(* CoDeSys 2.3.9.31 project: X758PLC.pro *)
(* Libraries: TcBase.lib 14.5.09 11:14:08, TcSystem.lib 27.2.12 14:08:36, TcBaseMath.lib 27.7.04 11:07:56, TcMath.lib 23.9.04 14:15:30, TcMC2.lib 23.8.12 10:01:14, STANDARD.LIB 5.6.98 11:03:02 *)

(* Task configuration *)
TASK Standard (PRIORITY := 0, INTERVAL := T#10ms);
	MAIN
END_TASK

(* Global variable list: Global_Variables *)
VAR_GLOBAL
	Axis_X	:	Axis_Ref;
	Axis_Y	:	Axis_Ref;
	Axis_F	:	Axis_Ref;
	Axis_T	:	Axis_Ref;
END_VAR

(* Global variable list: TwinCAT_Configuration *)
(* Generated automatically by TwinCAT - (read only) *)
VAR_CONFIG
	MAIN.BFI1 AT %IX512.0 : BOOL;	(*  ~ {LinkedWith:TIID^Device 2 (EtherCAT)^Term 1 (EK1100)^Term 2 (EL1889)^Channel 1^Input} *)
	MAIN.BFI2 AT %IX512.1 : BOOL;	(*  ~ {LinkedWith:TIID^Device 2 (EtherCAT)^Term 1 (EK1100)^Term 2 (EL1889)^Channel 2^Input} *)
	MAIN.BFI3 AT %IX512.2 : BOOL;	(*  ~ {LinkedWith:TIID^Device 2 (EtherCAT)^Term 1 (EK1100)^Term 2 (EL1889)^Channel 3^Input} *)
	MAIN.BFI4 AT %IX512.3 : BOOL;	(*  ~ {LinkedWith:TIID^Device 2 (EtherCAT)^Term 1 (EK1100)^Term 2 (EL1889)^Channel 4^Input} *)
	MAIN.BFI5 AT %IX512.4 : BOOL;	(*  ~ {LinkedWith:TIID^Device 2 (EtherCAT)^Term 1 (EK1100)^Term 2 (EL1889)^Channel 5^Input} *)
	MAIN.BFI6 AT %IX512.5 : BOOL;	(*  ~ {LinkedWith:TIID^Device 2 (EtherCAT)^Term 1 (EK1100)^Term 2 (EL1889)^Channel 6^Input} *)
	MAIN.BFI7 AT %IX512.6 : BOOL;	(*  ~ {LinkedWith:TIID^Device 2 (EtherCAT)^Term 1 (EK1100)^Term 2 (EL1889)^Channel 7^Input} *)
	MAIN.BFI8 AT %IX516.0 : BOOL;
	MAIN.BFI9 AT %IX516.1 : BOOL;
	MAIN.BFO1 AT %QX512.0 : BOOL;	(*  ~ {LinkedWith:TIID^Device 2 (EtherCAT)^Term 1 (EK1100)^Term 3 (EL2889)^Channel 1^Output} *)
	MAIN.BFO2 AT %QX512.1 : BOOL;	(*  ~ {LinkedWith:TIID^Device 2 (EtherCAT)^Term 1 (EK1100)^Term 3 (EL2889)^Channel 2^Output} *)
	MAIN.BFO3 AT %QX512.2 : BOOL;	(*  ~ {LinkedWith:TIID^Device 2 (EtherCAT)^Term 1 (EK1100)^Term 3 (EL2889)^Channel 3^Output} *)
	.Axis_X.PlcToNc AT %QB0 : PLCTONC_AXIS_REF;	(*  ~ {LinkedWith:TINC^NC-Task 1 SAF^Axes^Axis 1^Inputs^Axis 1_FromPlc} *)
	.Axis_X.NcToPlc AT %IB0 : NCTOPLC_AXIS_REF;	(*  ~ {LinkedWith:TINC^NC-Task 1 SAF^Axes^Axis 1^Outputs^Axis 1_ToPlc} *)
	.Axis_Y.PlcToNc AT %QB128 : PLCTONC_AXIS_REF;	(*  ~ {LinkedWith:TINC^NC-Task 1 SAF^Axes^Axis 2^Inputs^Axis 2_FromPlc} *)
	.Axis_Y.NcToPlc AT %IB128 : NCTOPLC_AXIS_REF;	(*  ~ {LinkedWith:TINC^NC-Task 1 SAF^Axes^Axis 2^Outputs^Axis 2_ToPlc} *)
	.Axis_F.PlcToNc AT %QB256 : PLCTONC_AXIS_REF;	(*  ~ {LinkedWith:TINC^NC-Task 1 SAF^Axes^Axis 3^Inputs^Axis 3_FromPlc} *)
	.Axis_F.NcToPlc AT %IB256 : NCTOPLC_AXIS_REF;	(*  ~ {LinkedWith:TINC^NC-Task 1 SAF^Axes^Axis 3^Outputs^Axis 3_ToPlc} *)
	.Axis_T.PlcToNc AT %QB384 : PLCTONC_AXIS_REF;	(*  ~ {LinkedWith:TINC^NC-Task 1 SAF^Axes^Axis 4^Inputs^Axis 4_FromPlc} *)
	.Axis_T.NcToPlc AT %IB384 : NCTOPLC_AXIS_REF;	(*  ~ {LinkedWith:TINC^NC-Task 1 SAF^Axes^Axis 4^Outputs^Axis 4_ToPlc} *)
END_VAR

(* POU MAIN, SFC *)
PROGRAM MAIN
VAR
	SFCInit: BOOL;	(* SFC流程控制标志位 *)
	SFCReset: BOOL;	(* SFC流程控制标志位 *)

	Trans1: BOOL;
	Trans2: BOOL;
	Trans3: BOOL;
	Trans4: BOOL;
	Trans5: BOOL;
	Trans6: BOOL;
	Trans7: BOOL;	(*  *)
	Trans8: BOOL;
	Trans9: BOOL;
	Trans10: BOOL;
	Trans11: BOOL;

	PowerAction1: MC_Power;
	PowerAction2: MC_Power;
	PowerAction3: MC_Power;
	PowerAction4: MC_Power;


	E1: BOOL;


	PowerOn1: BOOL;
	PowerOn2: BOOL;
	PowerOn3: BOOL;	(* 伺服ON标志 *)
	PowerOn4: BOOL;

	E2: BOOL;
	ResetAction1: MC_Reset;
	E3: BOOL;
	E4: BOOL;
	MoveAbsolute1: MC_MoveAbsolute;
	E5: BOOL;
	P1: LREAL;
	V1: LREAL;
	E6: BOOL;
	Jog1: MC_Jog;
	E7: BOOL;
	E8: BOOL;

	F1: BOOL;
	F2: BOOL;
	ResetAction2: MC_Reset;
	F3: BOOL;
	F4: BOOL;
	F5: BOOL;
	MoveAbsolute2: MC_MoveAbsolute;
	P2: LREAL;
	V2: LREAL;
	F6: BOOL;
	Jog2: MC_Jog;
	F8: BOOL;
	F7: BOOL;
	G1: BOOL;
	G2: BOOL;
	ResetAction3: MC_Reset;
	G3: BOOL;
	G4: BOOL;
	MoveAbsolute3: MC_MoveAbsolute;
	P3: LREAL;
	V3: LREAL;
	G5: BOOL;
	G6: BOOL;
	Jog3: MC_Jog;
	G7: BOOL;
	G8: BOOL;
	E9: BOOL;
	Home1: MC_Home;
	BFI1 AT %I*	:	BOOL;
	BFI2 AT %I*	:	BOOL;
	BFI3 AT %I*	:	BOOL;
	BFI4 AT %I*	:	BOOL;
	BFI5 AT %I*	:	BOOL;
	BFI6 AT %I*	:	BOOL;
	BFI7 AT %I*	:	BOOL;
	BFI8 AT %I*	:	BOOL;
	BFI9 AT %I*	:	BOOL;

	BFO1 AT %Q*	:	BOOL;
	BFO2 AT %Q*	:	BOOL;
	BFO3 AT %Q*	:	BOOL;
	F9: BOOL;
	Home2: MC_Home;
	F10: BOOL;
	E10: BOOL;
	G9: BOOL;
	Home3: MC_Home;
	G10: BOOL;
	H1: BOOL;
	H2: BOOL;
	ResetAction4: MC_Reset;
	H3: BOOL;
	H4: BOOL;
	MoveAbsolute4: MC_MoveAbsolute;
	H5: BOOL;
	P4: LREAL;
	V4: LREAL;
	H6: BOOL;
	H7: BOOL;
	Jog4: MC_Jog;
	H8: BOOL;
	H9: BOOL;
	Home4: MC_Home;
	H10: BOOL;

	XRDY	:	BOOL;
	YRDY	:	BOOL;
	FRDY	:	BOOL;
	TRDY	:	BOOL;

	EF0: BOOL;
	EF1: BOOL;
	EF2: BOOL;
	EF3: BOOL;
	TON1: TON;
	EF4: BOOL;
	TON2: TON;
	EF5: BOOL;
	EF6: BOOL;
	E11: BOOL;
	Stop1: MC_Stop;
	E12: BOOL;
	F11: BOOL;
	F12: BOOL;
	Stop2: MC_Stop;
	G11: BOOL;
	Stop3: MC_Stop;
	G12: BOOL;
	H11: BOOL;
	Stop4: MC_Stop;
	H12: BOOL;
	EF7: BOOL;
	F100: BOOL;
	F101: BOOL;
	F102: BOOL;
	TON3: TON;
	F103: BOOL;
	F104: BOOL;
	F105: BOOL;
	T100: BOOL;
	T101: BOOL;
	T102: BOOL;
	TON4: TON;

	T103: BOOL;

	T104: BOOL;
	T105: BOOL;
	UnloadCMD: BOOL;
	EF10: BOOL;
	EF11: BOOL;
	EF12: BOOL;
	EF13: BOOL;
	EF14: BOOL;
	TON5: TON;
	EF15: BOOL;
	TON6: TON;
	EF16: BOOL;
	TON7: TON;
	EF17: BOOL;
	EF18: BOOL;
	EF19: BOOL;
	EF20: BOOL;
	EF21: BOOL;
	EF22: BOOL;
	EF23: BOOL;
	EF24: BOOL;
	TON8: TON;
	EF25: BOOL;
	TON9: TON;
	EF26: BOOL;
	TON10: TON;
	EF27: BOOL;
	EF28: BOOL;
	EF29: BOOL;
	EF30: BOOL;
	XYDebugCMD: BOOL;
	XYDebugComplete: BOOL;
END_VAR
VAR PERSISTENT
	Override1: UINT;	(* 功率 *)
	Override2: UINT;
	Override3: UINT;
	Override4: UINT;

	PickPositionX	:	LREAL;
	PickPositionY	:	LREAL;
	RunVelocityX	:	LREAL;
	RunVelocityY	:	LREAL;

	InitPositionF	:	LREAL;
	RunVelocityF	:	LREAL;

	TransPositionT1	:	LREAL;
	RunVelocityT	:	LREAL;

	ReleasePositionXY	:	ARRAY	[0..11,0..1]	OF	LREAL;
	XYIndex	:	INT;

	ReleasePositionX1	:	LREAL;
	ReleasePositionY1	:	LREAL;
	ReleasePositionX2	:	LREAL;
	ReleasePositionY2	:	LREAL;
	ReleasePositionX3	:	LREAL;
	ReleasePositionY3	:	LREAL;
	DeltaX	:	LREAL;
	DeltaY	:	LREAL;


	Calc_i	:	INT;
	Calc_Start	:	BOOL;





END_VAR
VAR (* helpers for the ST form of the networks *)
	_p1 : BOOL;
	_p2 : BOOL;
	_p3 : BOOL;
	_p4 : BOOL;
	_p5 : BOOL;
	_p6 : BOOL;
	_p7 : BOOL;
	_p8 : BOOL;
	_p9 : BOOL;
	_p10 : BOOL;
	_p11 : BOOL;
	_p12 : BOOL;
	_p13 : BOOL;
	_p14 : BOOL;
	_p15 : BOOL;
	_p16 : BOOL;
	_p17 : BOOL;
	_p18 : BOOL;
	_p19 : BOOL;
	_p20 : BOOL;
	_p21 : BOOL;
	_p22 : BOOL;
	_p23 : BOOL;
	_p24 : BOOL;
	_p25 : BOOL;
	_p26 : BOOL;
	_p27 : BOOL;
	_p28 : BOOL;
	_p29 : BOOL;
	_p30 : BOOL;
	_p31 : BOOL;
	_p32 : BOOL;
	_p33 : BOOL;
	_p34 : BOOL;
END_VAR
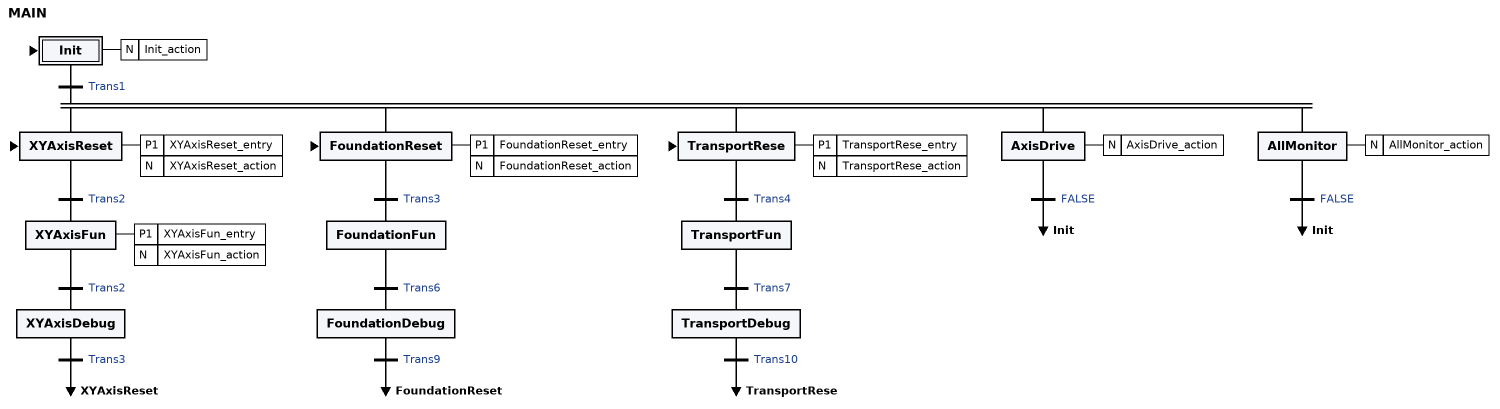
INITIAL_STEP Init:
	Init_action(N);
END_STEP
TRANSITION FROM Init TO (XYAxisReset, FoundationReset, TransportRese, AxisDrive, AllMonitor) := Trans1;
END_TRANSITION
STEP XYAxisReset:
	XYAxisReset_entry(P1);
	XYAxisReset_action(N);
END_STEP
TRANSITION FROM XYAxisReset TO XYAxisFun := Trans2;
END_TRANSITION
STEP XYAxisFun:
	XYAxisFun_entry(P1);
	XYAxisFun_action(N);
END_STEP
TRANSITION FROM XYAxisFun TO XYAxisDebug := Trans2;
END_TRANSITION
STEP XYAxisDebug:
END_STEP
TRANSITION FROM XYAxisDebug TO XYAxisReset := Trans3;
END_TRANSITION
STEP FoundationReset:
	FoundationReset_entry(P1);
	FoundationReset_action(N);
END_STEP
TRANSITION FROM FoundationReset TO FoundationFun := Trans3;
END_TRANSITION
STEP FoundationFun:
END_STEP
TRANSITION FROM FoundationFun TO FoundationDebug := Trans6;
END_TRANSITION
STEP FoundationDebug:
END_STEP
TRANSITION FROM FoundationDebug TO FoundationReset := Trans9;
END_TRANSITION
STEP TransportRese:
	TransportRese_entry(P1);
	TransportRese_action(N);
END_STEP
TRANSITION FROM TransportRese TO TransportFun := Trans4;
END_TRANSITION
STEP TransportFun:
END_STEP
TRANSITION FROM TransportFun TO TransportDebug := Trans7;
END_TRANSITION
STEP TransportDebug:
END_STEP
TRANSITION FROM TransportDebug TO TransportRese := Trans10;
END_TRANSITION
STEP AxisDrive:
	AxisDrive_action(N);
END_STEP
TRANSITION FROM AxisDrive TO Init := FALSE;
END_TRANSITION
STEP AllMonitor:
	AllMonitor_action(N);
END_STEP
TRANSITION FROM AllMonitor TO Init := FALSE;
END_TRANSITION

ACTION Init_action:
;
END_ACTION

ACTION XYAxisReset_entry:
EF0	:=	TRUE;
END_ACTION

ACTION XYAxisReset_action:
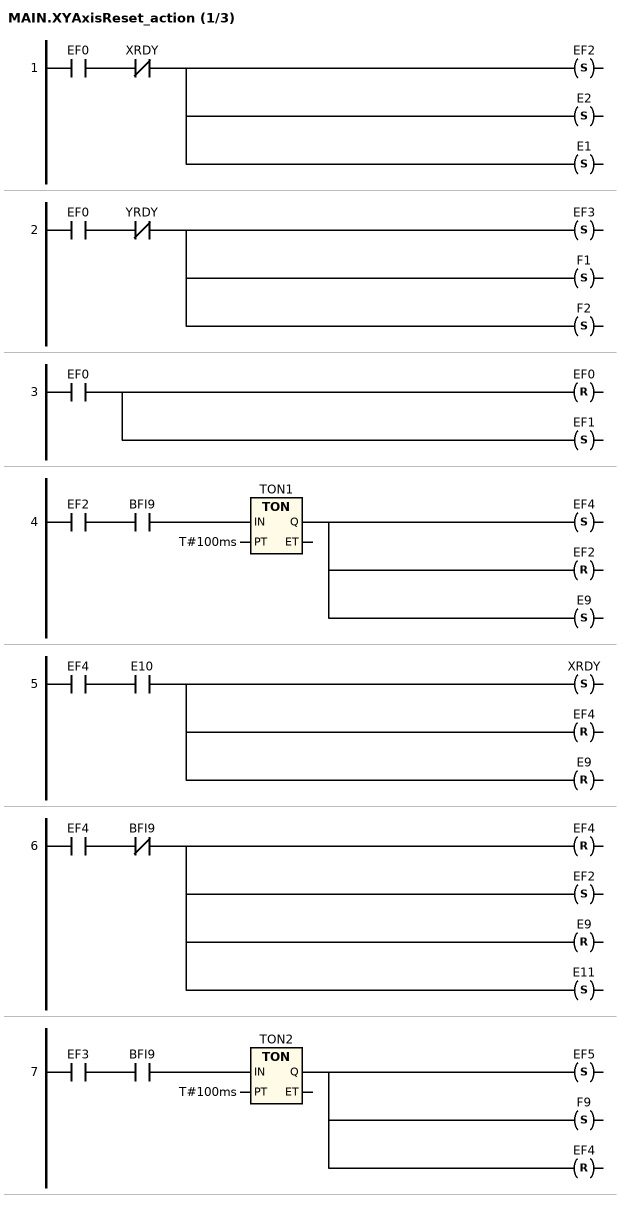
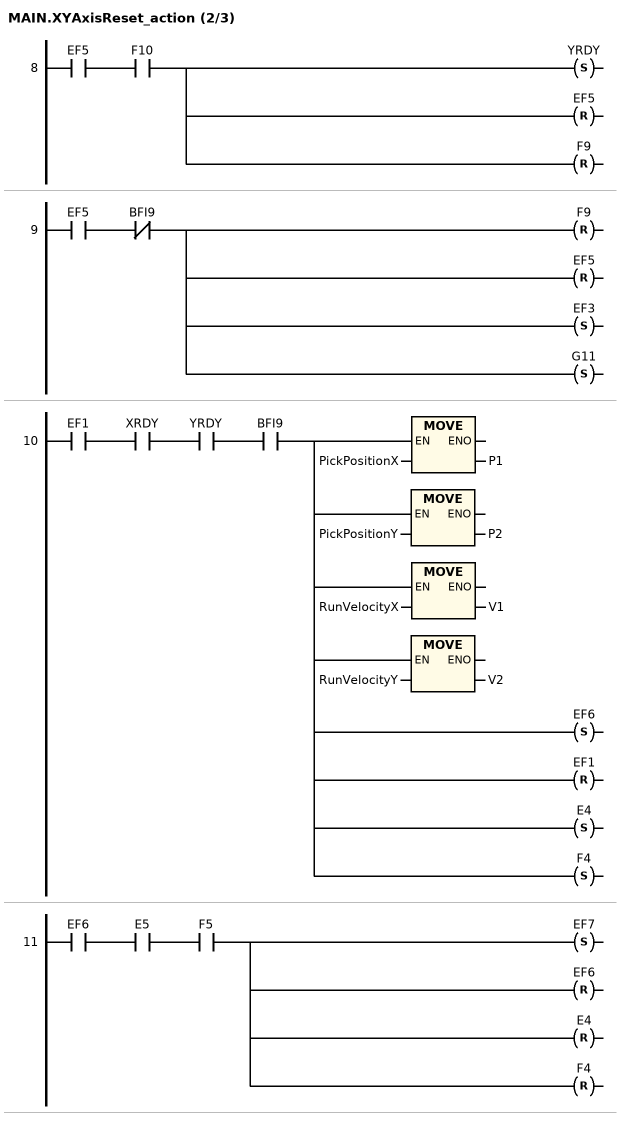
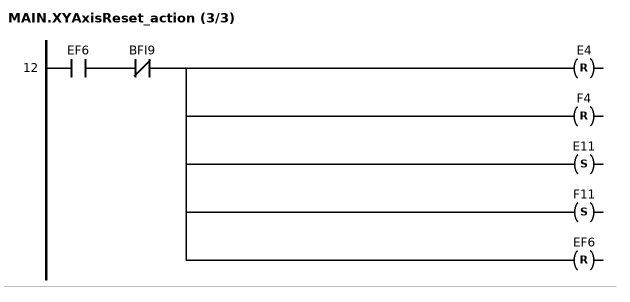
_LD_ (* Ladder Diagram *)
NETWORK 1
	[EF0] - [/XRDY] --- (S EF2) (S E2) (S E1)
NETWORK 2
	[EF0] - [/YRDY] --- (S EF3) (S F1) (S F2)
NETWORK 3
	[EF0] --- (R EF0) (S EF1)
NETWORK 4
	[EF2] - [BFI9] - TON1:TON(IN: *, PT: T#100ms) --- (S EF4) (R EF2) (S E9)
NETWORK 5
	[EF4] - [E10] --- (S XRDY) (R EF4) (R E9)
NETWORK 6
	[EF4] - [/BFI9] --- (R EF4) (S EF2) (R E9) (S E11)
NETWORK 7
	[EF3] - [BFI9] - TON2:TON(IN: *, PT: T#100ms) --- (S EF5) (S F9) (R EF4)
NETWORK 8
	[EF5] - [F10] --- (S YRDY) (R EF5) (R F9)
NETWORK 9
	[EF5] - [/BFI9] --- (R F9) (R EF5) (S EF3) (S G11)
NETWORK 10
	[EF1] - [XRDY] - [YRDY] - [BFI9] --- (S EF6) (R EF1) (S E4) (S F4)
		EN --- MOVE(PickPositionX) => P1
		EN --- MOVE(PickPositionY) => P2
		EN --- MOVE(RunVelocityX) => V1
		EN --- MOVE(RunVelocityY) => V2
NETWORK 11
	[EF6] - [E5] - [F5] --- (S EF7) (R EF6) (R E4) (R F4)
NETWORK 12
	[EF6] - [/BFI9] --- (R E4) (R F4) (S E11) (S F11) (R EF6)
_END_LD_
(* the same logic as Structured Text *)
(* Network 1 *)
IF EF0 AND NOT XRDY THEN EF2 := TRUE; E2 := TRUE; E1 := TRUE; END_IF;
(* Network 2 *)
IF EF0 AND NOT YRDY THEN EF3 := TRUE; F1 := TRUE; F2 := TRUE; END_IF;
(* Network 3 *)
_p1 := EF0;
IF _p1 THEN EF0 := FALSE; EF1 := TRUE; END_IF;
(* Network 4 *)
TON1(IN := EF2 AND BFI9, PT := T#100ms);
IF TON1.Q THEN EF4 := TRUE; EF2 := FALSE; E9 := TRUE; END_IF;
(* Network 5 *)
_p2 := EF4 AND E10;
IF _p2 THEN XRDY := TRUE; EF4 := FALSE; E9 := FALSE; END_IF;
(* Network 6 *)
_p3 := EF4 AND NOT BFI9;
IF _p3 THEN EF4 := FALSE; EF2 := TRUE; E9 := FALSE; E11 := TRUE; END_IF;
(* Network 7 *)
TON2(IN := EF3 AND BFI9, PT := T#100ms);
IF TON2.Q THEN EF5 := TRUE; F9 := TRUE; EF4 := FALSE; END_IF;
(* Network 8 *)
_p4 := EF5 AND F10;
IF _p4 THEN YRDY := TRUE; EF5 := FALSE; F9 := FALSE; END_IF;
(* Network 9 *)
_p5 := EF5 AND NOT BFI9;
IF _p5 THEN F9 := FALSE; EF5 := FALSE; EF3 := TRUE; G11 := TRUE; END_IF;
(* Network 10 *)
_p6 := EF1 AND XRDY AND YRDY AND BFI9;
IF _p6 THEN
	P1 := PickPositionX;
	P2 := PickPositionY;
	V1 := RunVelocityX;
	V2 := RunVelocityY;
END_IF;
IF _p6 THEN EF6 := TRUE; EF1 := FALSE; E4 := TRUE; F4 := TRUE; END_IF;
(* Network 11 *)
_p7 := EF6 AND E5 AND F5;
IF _p7 THEN EF7 := TRUE; EF6 := FALSE; E4 := FALSE; F4 := FALSE; END_IF;
(* Network 12 *)
_p8 := EF6 AND NOT BFI9;
IF _p8 THEN E4 := FALSE; F4 := FALSE; E11 := TRUE; F11 := TRUE; EF6 := FALSE; END_IF;
END_ACTION

ACTION XYAxisFun_entry:
EF7 := FALSE;
END_ACTION

ACTION XYAxisFun_action:
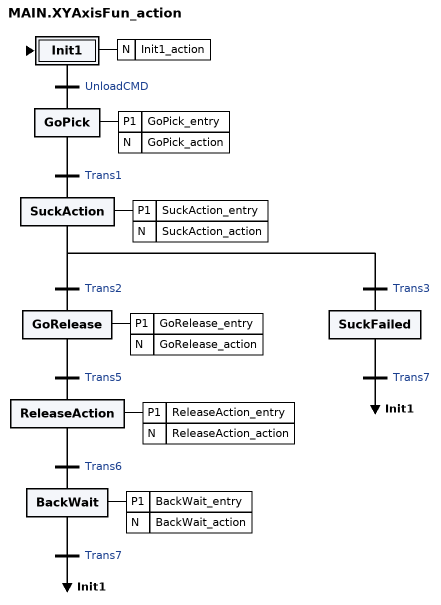
INITIAL_STEP Init1:
	Init1_action(N);
END_STEP
TRANSITION FROM Init1 TO GoPick := UnloadCMD;
END_TRANSITION
STEP GoPick:
	GoPick_entry(P1);
	GoPick_action(N);
END_STEP
TRANSITION FROM GoPick TO SuckAction := Trans1;
END_TRANSITION
STEP SuckAction:
	SuckAction_entry(P1);
	SuckAction_action(N);
END_STEP
TRANSITION FROM SuckAction TO GoRelease := Trans2;
END_TRANSITION
TRANSITION FROM SuckAction TO SuckFailed := Trans3;
END_TRANSITION
STEP SuckFailed:
END_STEP
TRANSITION FROM SuckFailed TO Init1 := Trans7;
END_TRANSITION
STEP GoRelease:
	GoRelease_entry(P1);
	GoRelease_action(N);
END_STEP
TRANSITION FROM GoRelease TO ReleaseAction := Trans5;
END_TRANSITION
STEP ReleaseAction:
	ReleaseAction_entry(P1);
	ReleaseAction_action(N);
END_STEP
TRANSITION FROM ReleaseAction TO BackWait := Trans6;
END_TRANSITION
STEP BackWait:
	BackWait_entry(P1);
	BackWait_action(N);
END_STEP
TRANSITION FROM BackWait TO Init1 := Trans7;
END_TRANSITION

ACTION Init1_action:
EF30 := FALSE;
END_ACTION

ACTION GoPick_entry:
UnloadCMD := FALSE;
EF10 := TRUE;
END_ACTION

ACTION GoPick_action:
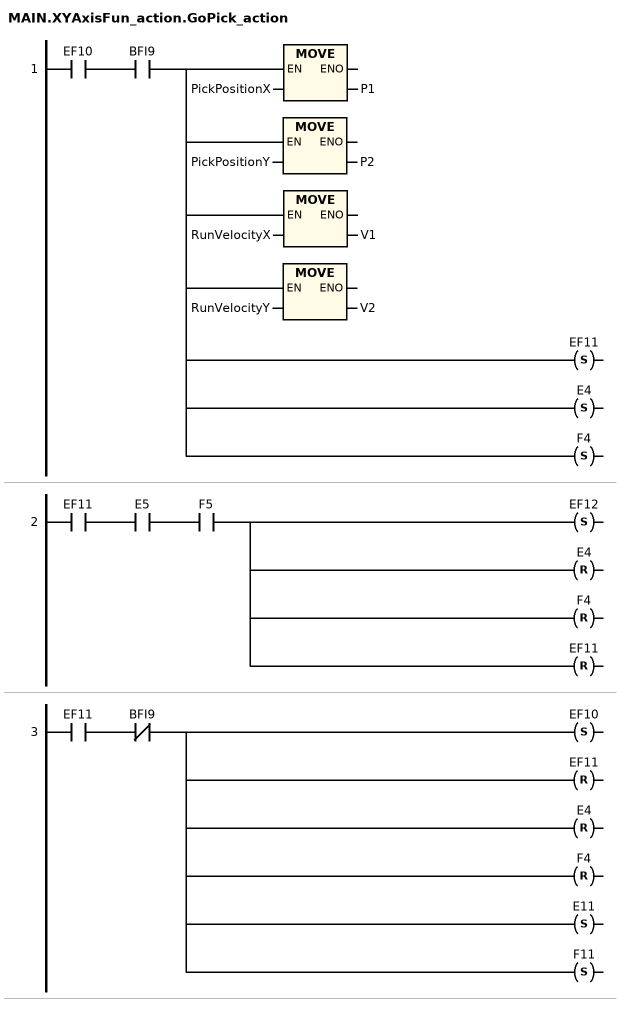
_LD_ (* Ladder Diagram *)
NETWORK 1
	[EF10] - [BFI9] --- (S EF11) (S E4) (S F4)
		EN --- MOVE(PickPositionX) => P1
		EN --- MOVE(PickPositionY) => P2
		EN --- MOVE(RunVelocityX) => V1
		EN --- MOVE(RunVelocityY) => V2
NETWORK 2
	[EF11] - [E5] - [F5] --- (S EF12) (R E4) (R F4) (R EF11)
NETWORK 3
	[EF11] - [/BFI9] --- (S EF10) (R EF11) (R E4) (R F4) (S E11) (S F11)
_END_LD_
(* the same logic as Structured Text *)
(* Network 1 *)
_p9 := EF10 AND BFI9;
IF _p9 THEN
	P1 := PickPositionX;
	P2 := PickPositionY;
	V1 := RunVelocityX;
	V2 := RunVelocityY;
END_IF;
IF _p9 THEN EF11 := TRUE; E4 := TRUE; F4 := TRUE; END_IF;
(* Network 2 *)
_p10 := EF11 AND E5 AND F5;
IF _p10 THEN EF12 := TRUE; E4 := FALSE; F4 := FALSE; EF11 := FALSE; END_IF;
(* Network 3 *)
_p11 := EF11 AND NOT BFI9;
IF _p11 THEN EF10 := TRUE; EF11 := FALSE; E4 := FALSE; F4 := FALSE; E11 := TRUE; F11 := TRUE; END_IF;
END_ACTION

ACTION SuckAction_entry:
EF12 := FALSE;
EF13 := TRUE;
END_ACTION

ACTION SuckAction_action:
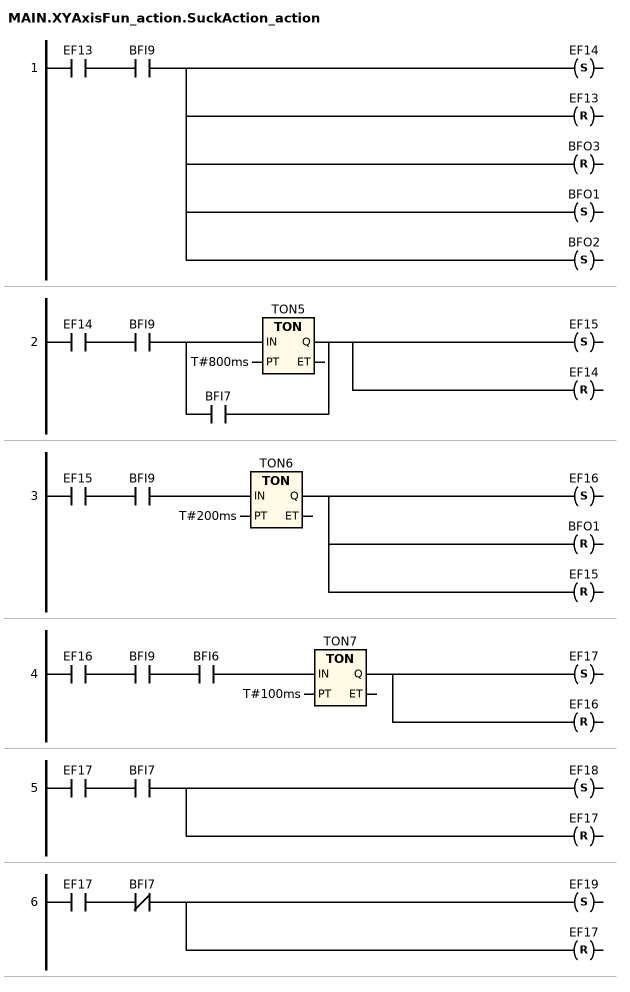
_LD_ (* Ladder Diagram *)
NETWORK 1
	[EF13] - [BFI9] --- (S EF14) (R EF13) (R BFO3) (S BFO1) (S BFO2)
NETWORK 2
	[EF14] - [BFI9] - { TON5:TON(IN: *, PT: T#800ms) | [BFI7] } --- (S EF15) (R EF14)
NETWORK 3
	[EF15] - [BFI9] - TON6:TON(IN: *, PT: T#200ms) --- (S EF16) (R BFO1) (R EF15)
NETWORK 4
	[EF16] - [BFI9] - [BFI6] - TON7:TON(IN: *, PT: T#100ms) --- (S EF17) (R EF16)
NETWORK 5
	[EF17] - [BFI7] --- (S EF18) (R EF17)
NETWORK 6
	[EF17] - [/BFI7] --- (S EF19) (R EF17)
_END_LD_
(* the same logic as Structured Text *)
(* Network 1 *)
_p12 := EF13 AND BFI9;
IF _p12 THEN EF14 := TRUE; EF13 := FALSE; BFO3 := FALSE; BFO1 := TRUE; BFO2 := TRUE; END_IF;
(* Network 2 *)
_p13 := EF14 AND BFI9;
TON5(IN := _p13, PT := T#800ms);
IF TON5.Q OR _p13 AND BFI7 THEN EF15 := TRUE; EF14 := FALSE; END_IF;
(* Network 3 *)
TON6(IN := EF15 AND BFI9, PT := T#200ms);
IF TON6.Q THEN EF16 := TRUE; BFO1 := FALSE; EF15 := FALSE; END_IF;
(* Network 4 *)
TON7(IN := EF16 AND BFI9 AND BFI6, PT := T#100ms);
IF TON7.Q THEN EF17 := TRUE; EF16 := FALSE; END_IF;
(* Network 5 *)
_p14 := EF17 AND BFI7;
IF _p14 THEN EF18 := TRUE; EF17 := FALSE; END_IF;
(* Network 6 *)
_p15 := EF17 AND NOT BFI7;
IF _p15 THEN EF19 := TRUE; EF17 := FALSE; END_IF;
END_ACTION

ACTION GoRelease_entry:
EF18 := FALSE;
EF20 := TRUE;
END_ACTION

ACTION GoRelease_action:
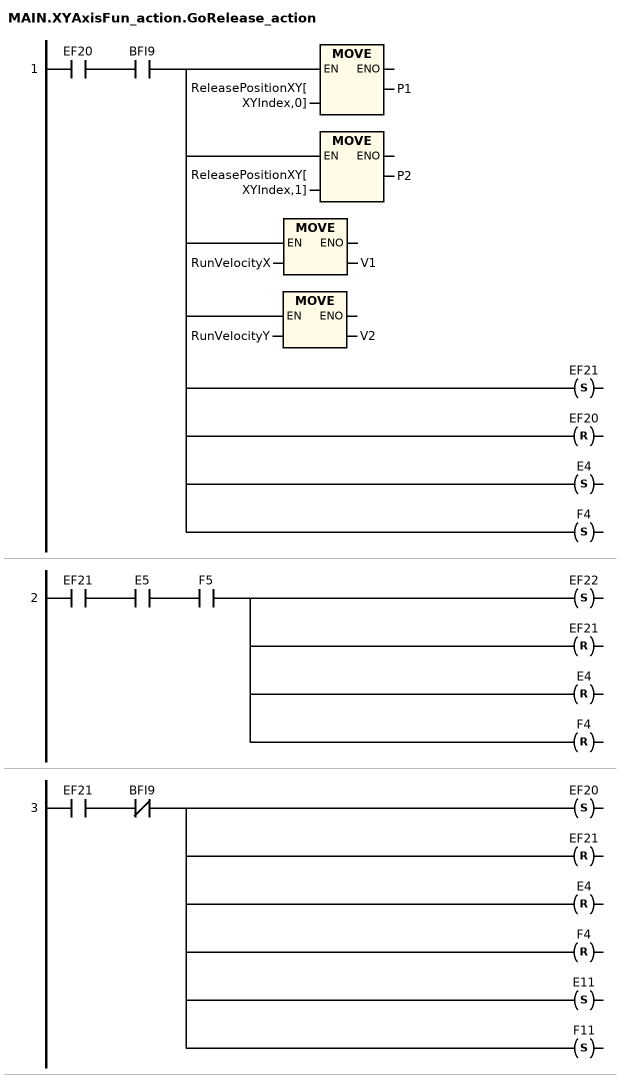
_LD_ (* Ladder Diagram *)
NETWORK 1
	[EF20] - [BFI9] --- (S EF21) (R EF20) (S E4) (S F4)
		EN --- MOVE(ReleasePositionXY[XYIndex,0]) => P1
		EN --- MOVE(ReleasePositionXY[XYIndex,1]) => P2
		EN --- MOVE(RunVelocityX) => V1
		EN --- MOVE(RunVelocityY) => V2
NETWORK 2
	[EF21] - [E5] - [F5] --- (S EF22) (R EF21) (R E4) (R F4)
NETWORK 3
	[EF21] - [/BFI9] --- (S EF20) (R EF21) (R E4) (R F4) (S E11) (S F11)
_END_LD_
(* the same logic as Structured Text *)
(* Network 1 *)
_p16 := EF20 AND BFI9;
IF _p16 THEN
	P1 := ReleasePositionXY[XYIndex,0];
	P2 := ReleasePositionXY[XYIndex,1];
	V1 := RunVelocityX;
	V2 := RunVelocityY;
END_IF;
IF _p16 THEN EF21 := TRUE; EF20 := FALSE; E4 := TRUE; F4 := TRUE; END_IF;
(* Network 2 *)
_p17 := EF21 AND E5 AND F5;
IF _p17 THEN EF22 := TRUE; EF21 := FALSE; E4 := FALSE; F4 := FALSE; END_IF;
(* Network 3 *)
_p18 := EF21 AND NOT BFI9;
IF _p18 THEN EF20 := TRUE; EF21 := FALSE; E4 := FALSE; F4 := FALSE; E11 := TRUE; F11 := TRUE; END_IF;
END_ACTION

ACTION ReleaseAction_entry:
EF22 := FALSE;
EF23 := TRUE;
END_ACTION

ACTION ReleaseAction_action:
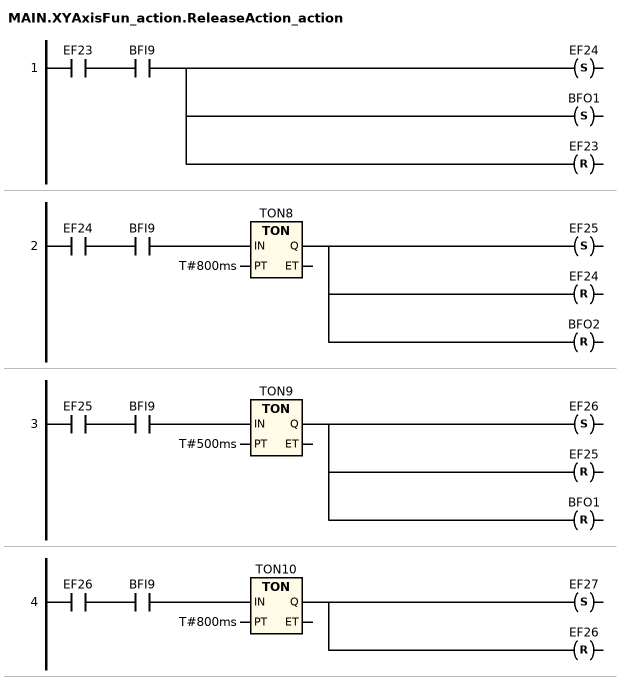
_LD_ (* Ladder Diagram *)
NETWORK 1
	[EF23] - [BFI9] --- (S EF24) (S BFO1) (R EF23)
NETWORK 2
	[EF24] - [BFI9] - TON8:TON(IN: *, PT: T#800ms) --- (S EF25) (R EF24) (R BFO2)
NETWORK 3
	[EF25] - [BFI9] - TON9:TON(IN: *, PT: T#500ms) --- (S EF26) (R EF25) (R BFO1)
NETWORK 4
	[EF26] - [BFI9] - TON10:TON(IN: *, PT: T#800ms) --- (S EF27) (R EF26)
_END_LD_
(* the same logic as Structured Text *)
(* Network 1 *)
_p19 := EF23 AND BFI9;
IF _p19 THEN EF24 := TRUE; BFO1 := TRUE; EF23 := FALSE; END_IF;
(* Network 2 *)
TON8(IN := EF24 AND BFI9, PT := T#800ms);
IF TON8.Q THEN EF25 := TRUE; EF24 := FALSE; BFO2 := FALSE; END_IF;
(* Network 3 *)
TON9(IN := EF25 AND BFI9, PT := T#500ms);
IF TON9.Q THEN EF26 := TRUE; EF25 := FALSE; BFO1 := FALSE; END_IF;
(* Network 4 *)
TON10(IN := EF26 AND BFI9, PT := T#800ms);
IF TON10.Q THEN EF27 := TRUE; EF26 := FALSE; END_IF;
END_ACTION

ACTION BackWait_entry:
EF27 := FALSE;
EF28 := TRUE;
END_ACTION

ACTION BackWait_action:
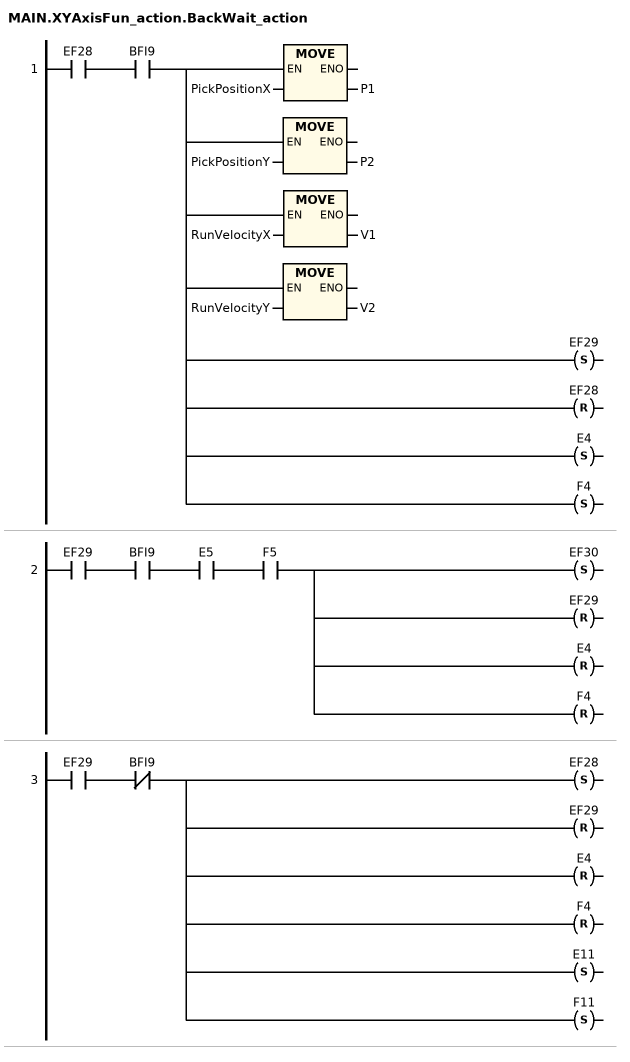
_LD_ (* Ladder Diagram *)
NETWORK 1
	[EF28] - [BFI9] --- (S EF29) (R EF28) (S E4) (S F4)
		EN --- MOVE(PickPositionX) => P1
		EN --- MOVE(PickPositionY) => P2
		EN --- MOVE(RunVelocityX) => V1
		EN --- MOVE(RunVelocityY) => V2
NETWORK 2
	[EF29] - [BFI9] - [E5] - [F5] --- (S EF30) (R EF29) (R E4) (R F4)
NETWORK 3
	[EF29] - [/BFI9] --- (S EF28) (R EF29) (R E4) (R F4) (S E11) (S F11)
_END_LD_
(* the same logic as Structured Text *)
(* Network 1 *)
_p20 := EF28 AND BFI9;
IF _p20 THEN
	P1 := PickPositionX;
	P2 := PickPositionY;
	V1 := RunVelocityX;
	V2 := RunVelocityY;
END_IF;
IF _p20 THEN EF29 := TRUE; EF28 := FALSE; E4 := TRUE; F4 := TRUE; END_IF;
(* Network 2 *)
_p21 := EF29 AND BFI9 AND E5 AND F5;
IF _p21 THEN EF30 := TRUE; EF29 := FALSE; E4 := FALSE; F4 := FALSE; END_IF;
(* Network 3 *)
_p22 := EF29 AND NOT BFI9;
IF _p22 THEN EF28 := TRUE; EF29 := FALSE; E4 := FALSE; F4 := FALSE; E11 := TRUE; F11 := TRUE; END_IF;
END_ACTION

TRANSITION Trans1:
_LD_ (* Ladder Diagram *)
NETWORK 1
	[EF12] - [BFI9]
_END_LD_
(* the same logic as Structured Text *)
(* Network 1 *)
Trans1 := EF12 AND BFI9;
END_TRANSITION

TRANSITION Trans2:
_LD_ (* Ladder Diagram *)
NETWORK 1
	[EF18] - [BFI9]
_END_LD_
(* the same logic as Structured Text *)
(* Network 1 *)
Trans2 := EF18 AND BFI9;
END_TRANSITION

TRANSITION Trans3:
_LD_ (* Ladder Diagram *)
NETWORK 1
	[EF19] - [BFI9]
_END_LD_
(* the same logic as Structured Text *)
(* Network 1 *)
Trans3 := EF19 AND BFI9;
END_TRANSITION

TRANSITION Trans7:
_LD_ (* Ladder Diagram *)
NETWORK 1
	*
_END_LD_
(* the same logic as Structured Text *)
(* Network 1 *)
Trans7 := TRUE;
END_TRANSITION

TRANSITION Trans5:
_LD_ (* Ladder Diagram *)
NETWORK 1
	[EF22] - [BFI9]
_END_LD_
(* the same logic as Structured Text *)
(* Network 1 *)
Trans5 := EF22 AND BFI9;
END_TRANSITION

TRANSITION Trans6:
_LD_ (* Ladder Diagram *)
NETWORK 1
	[EF27] - [BFI9]
_END_LD_
(* the same logic as Structured Text *)
(* Network 1 *)
Trans6 := EF27 AND BFI9;
END_TRANSITION

TRANSITION Trans7:
_LD_ (* Ladder Diagram *)
NETWORK 1
	[EF30] - [BFI9]
_END_LD_
(* the same logic as Structured Text *)
(* Network 1 *)
Trans7 := EF30 AND BFI9;
END_TRANSITION
END_ACTION

ACTION FoundationReset_entry:
F100 := TRUE;
END_ACTION

ACTION FoundationReset_action:
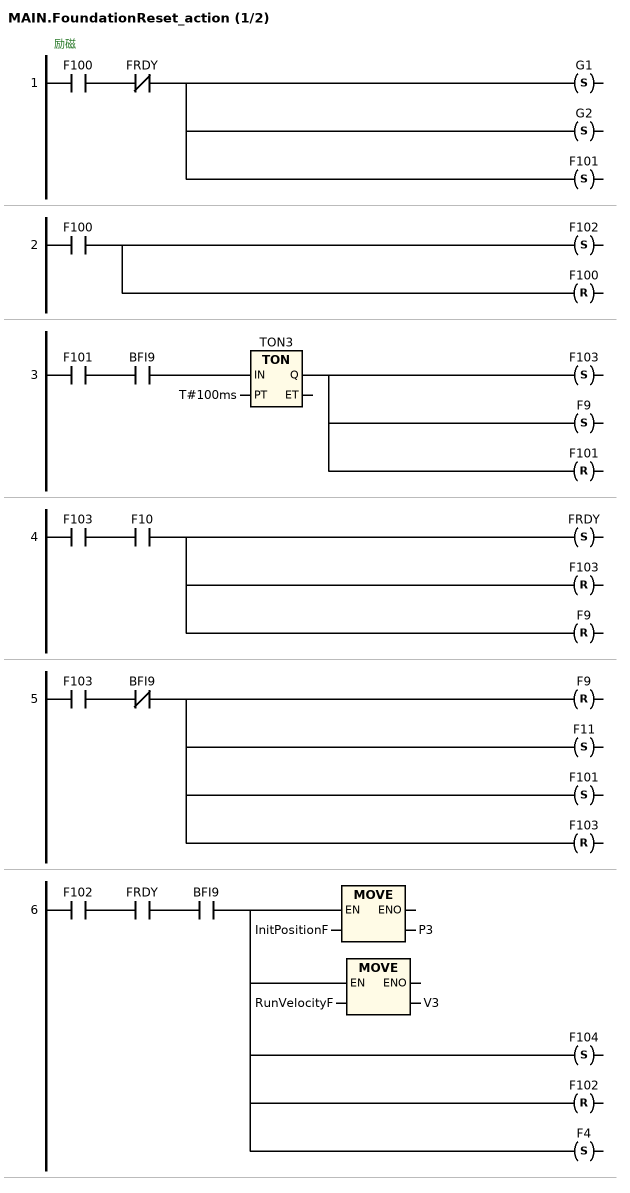
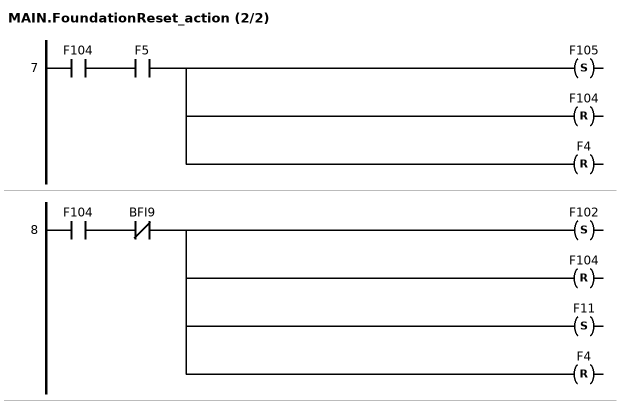
_LD_ (* Ladder Diagram *)
NETWORK 1 (* 励磁 *)
	[F100] - [/FRDY] --- (S G1) (S G2) (S F101)
NETWORK 2
	[F100] --- (S F102) (R F100)
NETWORK 3
	[F101] - [BFI9] - TON3:TON(IN: *, PT: T#100ms) --- (S F103) (S F9) (R F101)
NETWORK 4
	[F103] - [F10] --- (S FRDY) (R F103) (R F9)
NETWORK 5
	[F103] - [/BFI9] --- (R F9) (S F11) (S F101) (R F103)
NETWORK 6
	[F102] - [FRDY] - [BFI9] --- (S F104) (R F102) (S F4)
		EN --- MOVE(InitPositionF) => P3
		EN --- MOVE(RunVelocityF) => V3
NETWORK 7
	[F104] - [F5] --- (S F105) (R F104) (R F4)
NETWORK 8
	[F104] - [/BFI9] --- (S F102) (R F104) (S F11) (R F4)
_END_LD_
(* the same logic as Structured Text *)
(* Network 1: 励磁 *)
IF F100 AND NOT FRDY THEN G1 := TRUE; G2 := TRUE; F101 := TRUE; END_IF;
(* Network 2 *)
_p23 := F100;
IF _p23 THEN F102 := TRUE; F100 := FALSE; END_IF;
(* Network 3 *)
TON3(IN := F101 AND BFI9, PT := T#100ms);
IF TON3.Q THEN F103 := TRUE; F9 := TRUE; F101 := FALSE; END_IF;
(* Network 4 *)
_p24 := F103 AND F10;
IF _p24 THEN FRDY := TRUE; F103 := FALSE; F9 := FALSE; END_IF;
(* Network 5 *)
_p25 := F103 AND NOT BFI9;
IF _p25 THEN F9 := FALSE; F11 := TRUE; F101 := TRUE; F103 := FALSE; END_IF;
(* Network 6 *)
_p26 := F102 AND FRDY AND BFI9;
IF _p26 THEN
	P3 := InitPositionF;
	V3 := RunVelocityF;
END_IF;
IF _p26 THEN F104 := TRUE; F102 := FALSE; F4 := TRUE; END_IF;
(* Network 7 *)
_p27 := F104 AND F5;
IF _p27 THEN F105 := TRUE; F104 := FALSE; F4 := FALSE; END_IF;
(* Network 8 *)
_p28 := F104 AND NOT BFI9;
IF _p28 THEN F102 := TRUE; F104 := FALSE; F11 := TRUE; F4 := FALSE; END_IF;
END_ACTION

ACTION TransportRese_entry:
T100 := TRUE;
END_ACTION

ACTION TransportRese_action:
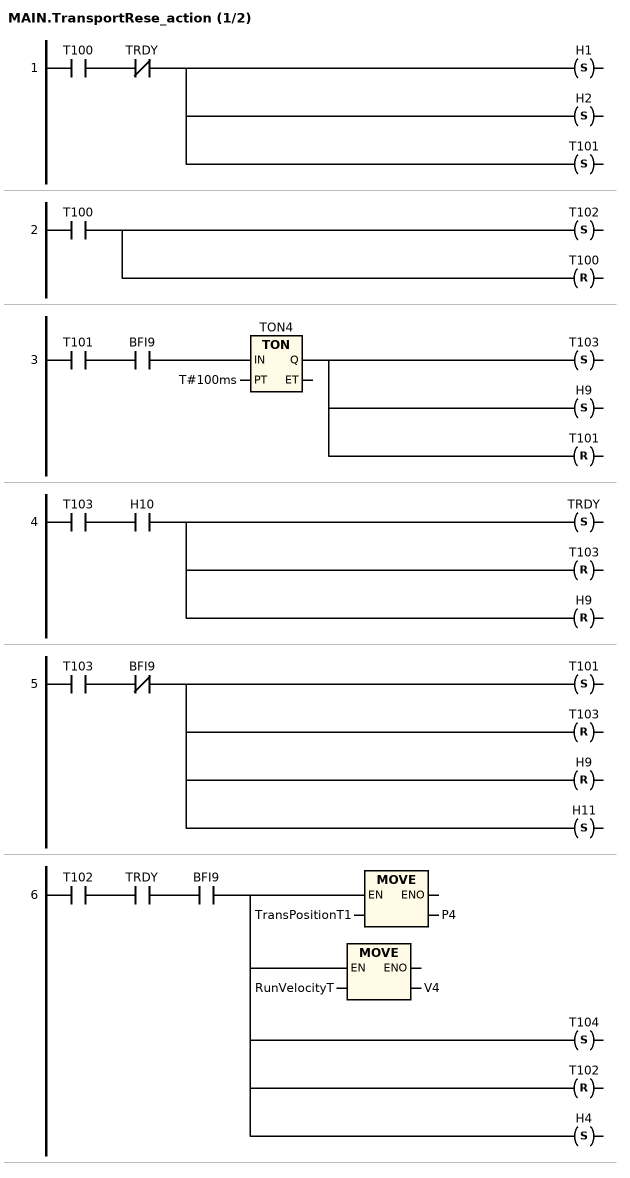
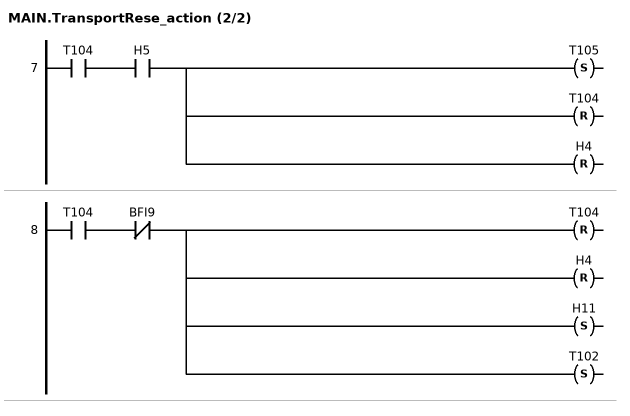
_LD_ (* Ladder Diagram *)
NETWORK 1
	[T100] - [/TRDY] --- (S H1) (S H2) (S T101)
NETWORK 2
	[T100] --- (S T102) (R T100)
NETWORK 3
	[T101] - [BFI9] - TON4:TON(IN: *, PT: T#100ms) --- (S T103) (S H9) (R T101)
NETWORK 4
	[T103] - [H10] --- (S TRDY) (R T103) (R H9)
NETWORK 5
	[T103] - [/BFI9] --- (S T101) (R T103) (R H9) (S H11)
NETWORK 6
	[T102] - [TRDY] - [BFI9] --- (S T104) (R T102) (S H4)
		EN --- MOVE(TransPositionT1) => P4
		EN --- MOVE(RunVelocityT) => V4
NETWORK 7
	[T104] - [H5] --- (S T105) (R T104) (R H4)
NETWORK 8
	[T104] - [/BFI9] --- (R T104) (R H4) (S H11) (S T102)
_END_LD_
(* the same logic as Structured Text *)
(* Network 1 *)
IF T100 AND NOT TRDY THEN H1 := TRUE; H2 := TRUE; T101 := TRUE; END_IF;
(* Network 2 *)
_p29 := T100;
IF _p29 THEN T102 := TRUE; T100 := FALSE; END_IF;
(* Network 3 *)
TON4(IN := T101 AND BFI9, PT := T#100ms);
IF TON4.Q THEN T103 := TRUE; H9 := TRUE; T101 := FALSE; END_IF;
(* Network 4 *)
_p30 := T103 AND H10;
IF _p30 THEN TRDY := TRUE; T103 := FALSE; H9 := FALSE; END_IF;
(* Network 5 *)
_p31 := T103 AND NOT BFI9;
IF _p31 THEN T101 := TRUE; T103 := FALSE; H9 := FALSE; H11 := TRUE; END_IF;
(* Network 6 *)
_p32 := T102 AND TRDY AND BFI9;
IF _p32 THEN
	P4 := TransPositionT1;
	V4 := RunVelocityT;
END_IF;
IF _p32 THEN T104 := TRUE; T102 := FALSE; H4 := TRUE; END_IF;
(* Network 7 *)
_p33 := T104 AND H5;
IF _p33 THEN T105 := TRUE; T104 := FALSE; H4 := FALSE; END_IF;
(* Network 8 *)
_p34 := T104 AND NOT BFI9;
IF _p34 THEN T104 := FALSE; H4 := FALSE; H11 := TRUE; T102 := TRUE; END_IF;
END_ACTION

ACTION AxisDrive_action:
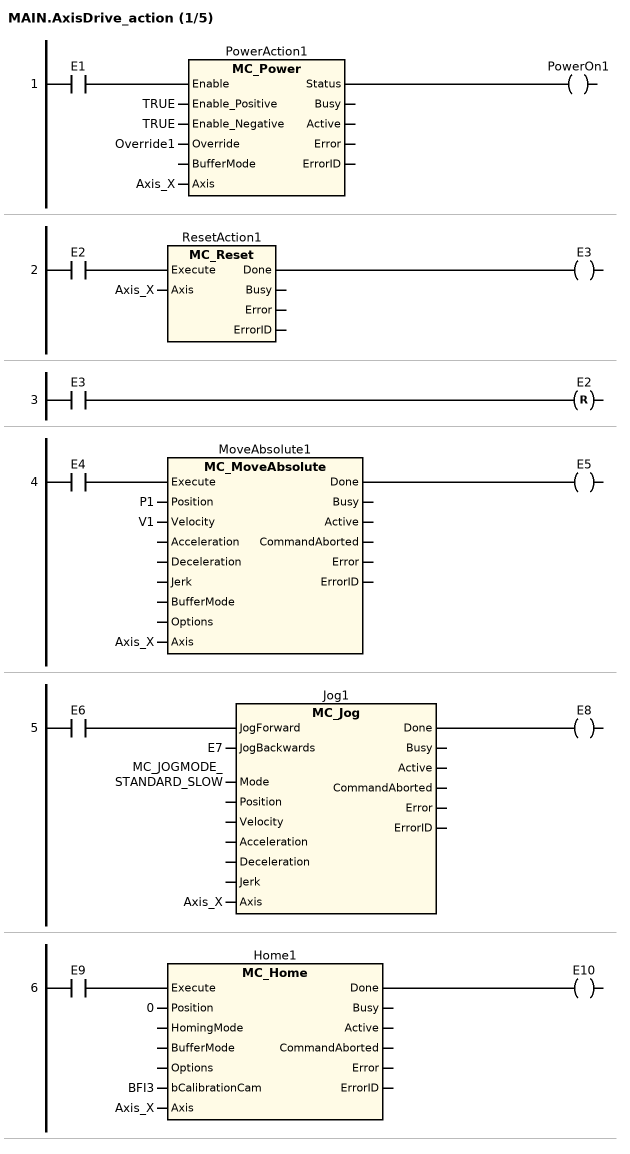
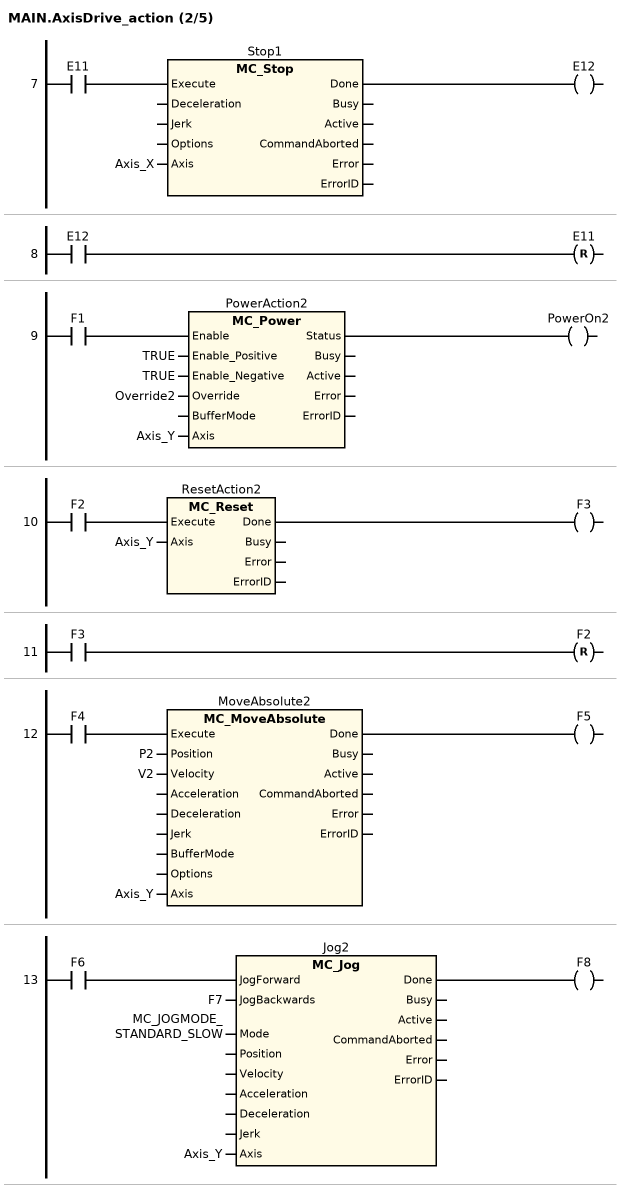
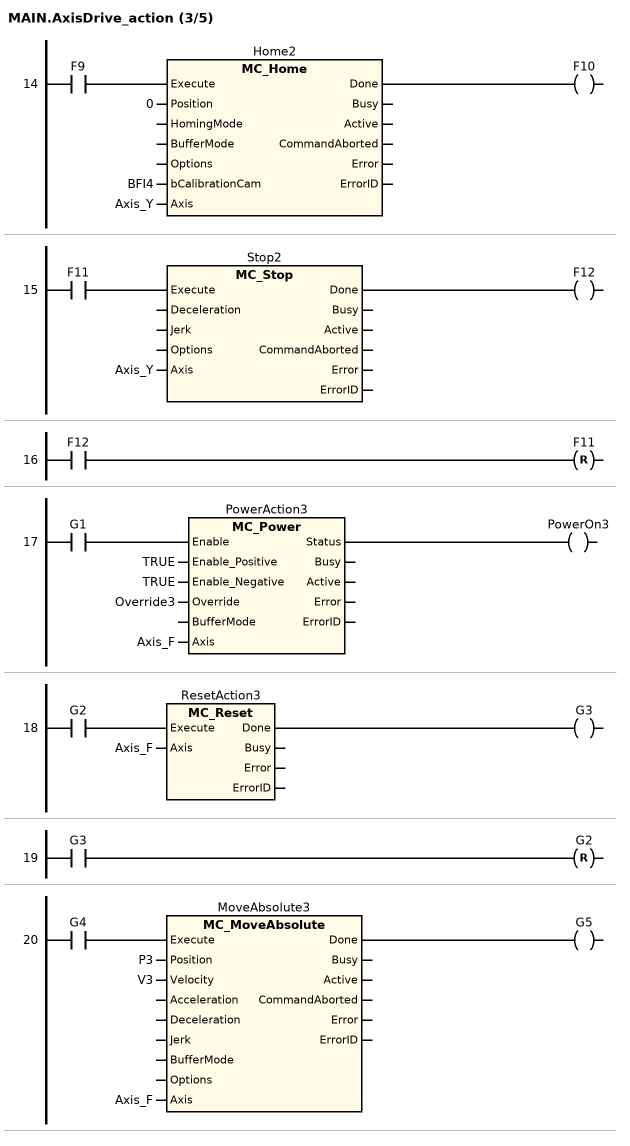
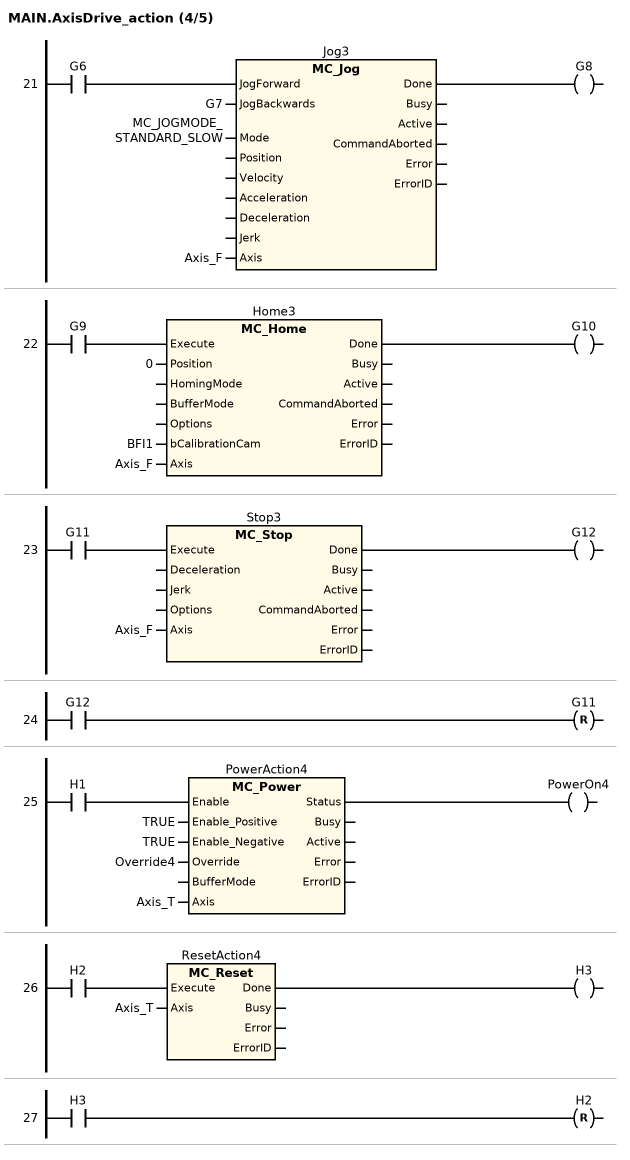
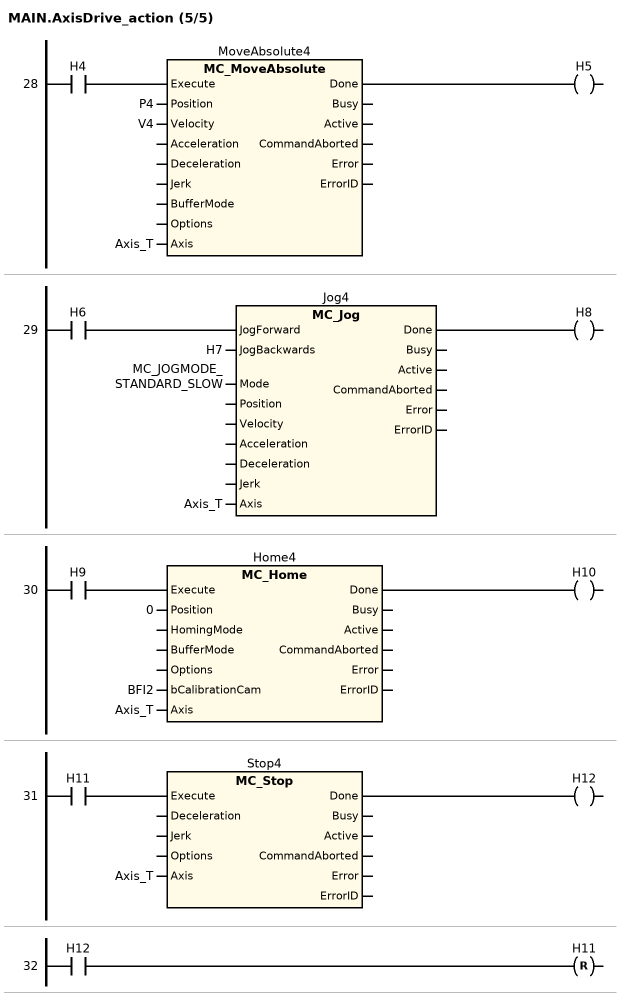
_LD_ (* Ladder Diagram *)
NETWORK 1
	[E1] - PowerAction1:MC_Power(Enable: *, Enable_Positive: TRUE, Enable_Negative: TRUE, Override: Override1, BufferMode: , Axis: Axis_X) --- (PowerOn1)
NETWORK 2
	[E2] - ResetAction1:MC_Reset(Execute: *, Axis: Axis_X) --- (E3)
NETWORK 3
	[E3] --- (R E2)
NETWORK 4
	[E4] - MoveAbsolute1:MC_MoveAbsolute(Execute: *, Position: P1, Velocity: V1, Acceleration: , Deceleration: , Jerk: , BufferMode: , Options: , Axis: Axis_X) --- (E5)
NETWORK 5
	[E6] - Jog1:MC_Jog(JogForward: *, JogBackwards: E7, Mode: MC_JOGMODE_STANDARD_SLOW, Position: , Velocity: , Acceleration: , Deceleration: , Jerk: , Axis: Axis_X) --- (E8)
NETWORK 6
	[E9] - Home1:MC_Home(Execute: *, Position: 0, HomingMode: , BufferMode: , Options: , bCalibrationCam: BFI3, Axis: Axis_X) --- (E10)
NETWORK 7
	[E11] - Stop1:MC_Stop(Execute: *, Deceleration: , Jerk: , Options: , Axis: Axis_X) --- (E12)
NETWORK 8
	[E12] --- (R E11)
NETWORK 9
	[F1] - PowerAction2:MC_Power(Enable: *, Enable_Positive: TRUE, Enable_Negative: TRUE, Override: Override2, BufferMode: , Axis: Axis_Y) --- (PowerOn2)
NETWORK 10
	[F2] - ResetAction2:MC_Reset(Execute: *, Axis: Axis_Y) --- (F3)
NETWORK 11
	[F3] --- (R F2)
NETWORK 12
	[F4] - MoveAbsolute2:MC_MoveAbsolute(Execute: *, Position: P2, Velocity: V2, Acceleration: , Deceleration: , Jerk: , BufferMode: , Options: , Axis: Axis_Y) --- (F5)
NETWORK 13
	[F6] - Jog2:MC_Jog(JogForward: *, JogBackwards: F7, Mode: MC_JOGMODE_STANDARD_SLOW, Position: , Velocity: , Acceleration: , Deceleration: , Jerk: , Axis: Axis_Y) --- (F8)
NETWORK 14
	[F9] - Home2:MC_Home(Execute: *, Position: 0, HomingMode: , BufferMode: , Options: , bCalibrationCam: BFI4, Axis: Axis_Y) --- (F10)
NETWORK 15
	[F11] - Stop2:MC_Stop(Execute: *, Deceleration: , Jerk: , Options: , Axis: Axis_Y) --- (F12)
NETWORK 16
	[F12] --- (R F11)
NETWORK 17
	[G1] - PowerAction3:MC_Power(Enable: *, Enable_Positive: TRUE, Enable_Negative: TRUE, Override: Override3, BufferMode: , Axis: Axis_F) --- (PowerOn3)
NETWORK 18
	[G2] - ResetAction3:MC_Reset(Execute: *, Axis: Axis_F) --- (G3)
NETWORK 19
	[G3] --- (R G2)
NETWORK 20
	[G4] - MoveAbsolute3:MC_MoveAbsolute(Execute: *, Position: P3, Velocity: V3, Acceleration: , Deceleration: , Jerk: , BufferMode: , Options: , Axis: Axis_F) --- (G5)
NETWORK 21
	[G6] - Jog3:MC_Jog(JogForward: *, JogBackwards: G7, Mode: MC_JOGMODE_STANDARD_SLOW, Position: , Velocity: , Acceleration: , Deceleration: , Jerk: , Axis: Axis_F) --- (G8)
NETWORK 22
	[G9] - Home3:MC_Home(Execute: *, Position: 0, HomingMode: , BufferMode: , Options: , bCalibrationCam: BFI1, Axis: Axis_F) --- (G10)
NETWORK 23
	[G11] - Stop3:MC_Stop(Execute: *, Deceleration: , Jerk: , Options: , Axis: Axis_F) --- (G12)
NETWORK 24
	[G12] --- (R G11)
NETWORK 25
	[H1] - PowerAction4:MC_Power(Enable: *, Enable_Positive: TRUE, Enable_Negative: TRUE, Override: Override4, BufferMode: , Axis: Axis_T) --- (PowerOn4)
NETWORK 26
	[H2] - ResetAction4:MC_Reset(Execute: *, Axis: Axis_T) --- (H3)
NETWORK 27
	[H3] --- (R H2)
NETWORK 28
	[H4] - MoveAbsolute4:MC_MoveAbsolute(Execute: *, Position: P4, Velocity: V4, Acceleration: , Deceleration: , Jerk: , BufferMode: , Options: , Axis: Axis_T) --- (H5)
NETWORK 29
	[H6] - Jog4:MC_Jog(JogForward: *, JogBackwards: H7, Mode: MC_JOGMODE_STANDARD_SLOW, Position: , Velocity: , Acceleration: , Deceleration: , Jerk: , Axis: Axis_T) --- (H8)
NETWORK 30
	[H9] - Home4:MC_Home(Execute: *, Position: 0, HomingMode: , BufferMode: , Options: , bCalibrationCam: BFI2, Axis: Axis_T) --- (H10)
NETWORK 31
	[H11] - Stop4:MC_Stop(Execute: *, Deceleration: , Jerk: , Options: , Axis: Axis_T) --- (H12)
NETWORK 32
	[H12] --- (R H11)
_END_LD_
(* the same logic as Structured Text *)
(* Network 1: see the listing above *)
(* Network 2 *)
ResetAction1(Execute := E2, Axis := Axis_X);
E3 := ResetAction1.Done;
(* Network 3 *)
IF E3 THEN E2 := FALSE; END_IF;
(* Network 4: see the listing above *)
(* Network 5: see the listing above *)
(* Network 6: see the listing above *)
(* Network 7: see the listing above *)
(* Network 8 *)
IF E12 THEN E11 := FALSE; END_IF;
(* Network 9: see the listing above *)
(* Network 10 *)
ResetAction2(Execute := F2, Axis := Axis_Y);
F3 := ResetAction2.Done;
(* Network 11 *)
IF F3 THEN F2 := FALSE; END_IF;
(* Network 12: see the listing above *)
(* Network 13: see the listing above *)
(* Network 14: see the listing above *)
(* Network 15: see the listing above *)
(* Network 16 *)
IF F12 THEN F11 := FALSE; END_IF;
(* Network 17: see the listing above *)
(* Network 18 *)
ResetAction3(Execute := G2, Axis := Axis_F);
G3 := ResetAction3.Done;
(* Network 19 *)
IF G3 THEN G2 := FALSE; END_IF;
(* Network 20: see the listing above *)
(* Network 21: see the listing above *)
(* Network 22: see the listing above *)
(* Network 23: see the listing above *)
(* Network 24 *)
IF G12 THEN G11 := FALSE; END_IF;
(* Network 25: see the listing above *)
(* Network 26 *)
ResetAction4(Execute := H2, Axis := Axis_T);
H3 := ResetAction4.Done;
(* Network 27 *)
IF H3 THEN H2 := FALSE; END_IF;
(* Network 28: see the listing above *)
(* Network 29: see the listing above *)
(* Network 30: see the listing above *)
(* Network 31: see the listing above *)
(* Network 32 *)
IF H12 THEN H11 := FALSE; END_IF;
END_ACTION

ACTION AllMonitor_action:
IF BFI8 THEN
	SFCReset := FALSE;
ELSE
	SFCReset := TRUE;
END_IF

IF Calc_Start THEN
	DeltaX := (ReleasePositionX3 - ReleasePositionX1)/3;
	DeltaY := (ReleasePositionY2 - ReleasePositionY1)/2;
	FOR Calc_i := 0 TO 11 DO
		ReleasePositionXY[Calc_i,0] := Calc_i/3*DeltaX + ReleasePositionX1;
		ReleasePositionXY[Calc_i,1] := (Calc_i MOD 3)*DeltaY + ReleasePositionY1;
	END_FOR
	Calc_Start := FALSE;
END_IF
END_ACTION

TRANSITION Trans1:
_LD_ (* Ladder Diagram *)
NETWORK 1
	[BFI8]
_END_LD_
(* the same logic as Structured Text *)
(* Network 1 *)
Trans1 := BFI8;
END_TRANSITION

TRANSITION Trans2:
_LD_ (* Ladder Diagram *)
NETWORK 1
	[EF7] - [BFI9]
_END_LD_
(* the same logic as Structured Text *)
(* Network 1 *)
Trans2 := EF7 AND BFI9;
END_TRANSITION

TRANSITION Trans2:
_LD_ (* Ladder Diagram *)
NETWORK 1
	[XYDebugCMD] - [INIT1]
_END_LD_
(* the same logic as Structured Text *)
(* Network 1 *)
Trans2 := XYDebugCMD AND INIT1;
END_TRANSITION

TRANSITION Trans3:
_LD_ (* Ladder Diagram *)
NETWORK 1
	[XYDebugComplete]
_END_LD_
(* the same logic as Structured Text *)
(* Network 1 *)
Trans3 := XYDebugComplete;
END_TRANSITION

TRANSITION Trans3:
_LD_ (* Ladder Diagram *)
NETWORK 1
	[F105]
_END_LD_
(* the same logic as Structured Text *)
(* Network 1 *)
Trans3 := F105;
END_TRANSITION

TRANSITION Trans4:
_LD_ (* Ladder Diagram *)
NETWORK 1
	[T105]
_END_LD_
(* the same logic as Structured Text *)
(* Network 1 *)
Trans4 := T105;
END_TRANSITION
END_PROGRAM
